//==================================================================================================
//							Beckhoff Automation Poland
//									23.11.2016
//			Bloczek do filtru inercyjnego do wygladzania przebiegow,					
//					czas próbkowania wyliczany wewnętrznie
//  v1.1	|| TC v 3.1.4020.28		|| - poprawienie inicjalizacji, notacja wegierska
// 	v1.0	|| TC v 3.1.4020.0		|| - pierwsza wersja
//==================================================================================================
FUNCTION_BLOCK FB_FilterEx_2
VAR_INPUT
	rIn										: REAL;					// Sygnal wejsciowy
	tTimeConstant							: TIME;					// Stala czasowa T gdy rOut = 0,63 * rIn 
END_VAR
VAR_OUTPUT
	rOut									: REAL;					// Przefiltrowany sygnal wyjsciowy, 
END_VAR
VAR
	rLastOut								: REAL;					// Wartosc wyjscia w poprzednim cyklu
	rCycleTime								: REAL; 				// [ms]
	rTimeConst								: REAL;					// [ms]
	tX										: TIME;					// Aktualny czas
	tY 										: TIME;					// Zmienna pomocnicza, poprzedni czas
	tCycleTime								: TIME;					// Wyliczony czas cyklu
	bFirstCycle								: BOOL := TRUE;			// Flaga pierwszego cyklu - nie mamy jeszce wyliczonego prawidlowo czasu cylu 
																	// - potrzebujemy dwoch cylki do odjecia czasu
END_VAR

// Obliczenie czasu cyklu do inkrementu
tX 					:= TIME();
IF NOT bFirstCycle THEN
	tCycleTime 		:= tX - tY;
END_IF
tY 					:= tX;
// Przeliczenie czasu na typ REAL
rCycleTime 			:= TIME_TO_REAL(tCycleTime);
rTimeConst 			:= TIME_TO_REAL(tTimeConstant);
// Wyliczenie wyjscia tylko jesli stala czasowa wieksza od 1 ms i zakonczylismy inicjalizacje
IF NOT bFirstCycle AND rTimeConst > 0.001 THEN
	rOut 			:= rLastOut + (rIn - rLastOut) * rCycleTime/rTimeConst;
	rLastOut 		:= rOut;
END_IF
// Zerowanie flagu pierwszego cyklu
bFirstCycle 		:= FALSE;

END_FUNCTION_BLOCK

(* stored: Version 1.2.0.0, ProductVersion 3.1.4026.13, FileIdentifier 2317ce36e7d1e832fbab9f84a441796fdd5a2529, FileSignature 7d8694e96052cf63b2681d5f0af7a2c03e3596a7d3a48a690e58171c0c68a8015cb998a34cf74543c571a50d6d7488fb4df590cf9e5306890d5573731a3418a1dcc77541924daa1a21ed8581e5c1c52246f57fb352bdfd6391dd307a41fb9759088fc3a62e529a081af468f02b4b6967ade1c81fba0b8850a8c0058f7d46d298f488884384f03b53817b79d152ff0294ddabe2784e8baf49cff4eca6f116aa6aa098f27bdd996082894b03adf04de800680e86824a8cf3ab10236d16cb8ff872fc94768fa9dfa7eb391a888815bda6087ce050da68a3fbba4fafb2b5e5c2347b0e1f45b2a71e73cd43d5ca22cda6d790a1cf31b513fde25e40bf8bfe55fa17e1
   POU FB_FilterEx_2: Id {077425bc-cdfc-4d8b-bbc0-07022d985fd2}, SpecialFunc None *)
